FUNCTION_BLOCK OrientStation
VAR_INPUT
	PrintStnADR	: UDINT;
END_VAR
VAR_OUTPUT
END_VAR
VAR
	rIO		: REFERENCE IO_Orient_typ;
	rStation : REFERENCE Station;
END_VAR

METHOD Cyclic : BOOL
VAR_INPUT
END_VAR
Station access PrintStnADR;
END_METHOD

END_FUNCTION_BLOCK

(* stored: Version 1.1.0.1, ProductVersion 3.1.4024.12
   POU OrientStation: Id {37722a1a-8fe0-0ed5-3944-0550e379750d}, SpecialFunc None
   Method Cyclic: Id {a820a9db-2ef7-0ad2-29be-a32b40c3d2e1} *)
